TYPE ST_PARAMETER_SELECTOR_STATE :
STRUCT
  AxisIndex   : UINT;             // what you selected mirrored back
  AxisId      : UDINT;            // matching Id to the index
  State       : ST_AXIS_STATE;    // result identifier to your command
  Info        : ST_NC_PARAMETER;  // read data
END_STRUCT
END_TYPE

(* stored: Version 1.1.0.1, ProductVersion 3.1.4026.18
   DUT ST_PARAMETER_SELECTOR_STATE: Id {39eac4db-60c2-4edc-99de-f5c8a822c18c} *)
